{attribute addProperty BoxType "EPP2817-0008-0016"}
{attribute addProperty Id "DIG_Diag_Inputs_ChannelAT %I*ARRAY[0..2] OF DIG_Diag_Inputs_Channel_AC4A9AF0192240DIG_Inputs_DeviceAT %I*DIG_Inputs_Device_2C95E2596480DIG_Output_ChannelAT %Q*ARRAY[0..2] OF DIG_Output_Channel_33B76376192240DIG_Outputs_DeviceAT %Q*DIG_Outputs_Device_735003021620WcStateAT %I*WcState_F855686C1620InfoDataAT %I*InfoData_BC63D37F80100"}
{attribute addProperty CRC "4293767907"}
{attribute addProperty SizeInBites "560"}
{attribute addProperty SizeInBytes "70"}
TYPE EPP2817_A6BB1E36 :
STRUCT
	{attribute addProperty Name "DIG_Diag_Inputs_Channel"}
	DIG_Diag_Inputs_Channel : ARRAY[0..2] OF DIG_Diag_Inputs_Channel_AC4A9AF0;
	{attribute addProperty Name "DIG_Inputs_Device"}
	DIG_Inputs_Device : DIG_Inputs_Device_2C95E259;
	{attribute addProperty Name "DIG_Output_Channel"}
	DIG_Output_Channel : ARRAY[0..2] OF DIG_Output_Channel_33B76376;
	{attribute addProperty Name "DIG_Outputs_Device"}
	DIG_Outputs_Device : DIG_Outputs_Device_73500302;
	{attribute addProperty Name "WcState"}
	WcState : WcState_F855686C;
	{attribute addProperty Name "InfoData"}
	InfoData : InfoData_BC63D37F;
END_STRUCT
END_TYPE

(* stored: Version 1.2.0.0, ProductVersion 3.1.4024.9
   DUT EPP2817_A6BB1E36: Id {e66cc0b8-7721-4673-95e0-4c2e0567793c} *)
